TYPE ST_ServoMove :
STRUCT
	Name : STRING(Param_Servo.DESCRIPTION_LEN) := 'Actuator'; //Name visualized on UI
	AdvanceFeedback_Used : BOOL;      //TRUE if advanced state feedback is used  
	RetractFeedback_Used  : BOOL;      //TRUE if retracted state feedback is used  
	AdvanceFeedbackTimeoutError : TIME; // How long we wait to see advanced feedback before we raise timeout error; 0 if not used
	RetractFeedbackTimeoutError : TIME; // How long we wait to see retracted feedback before we raise timeout error; 0 if not used
	SimFeedback_Advance_TimeElapsed : TIME; //If we do not use Advanced Feedback, serves as simulation delay after Advance Output is Set
	SimFeedback_Retract_TimeElapsed : TIME; //If we do not use Retracted Feedback, serves as simulation delay after Advance Output is Set
END_STRUCT
END_TYPE

(* stored: Version 1.1.0.1, ProductVersion 3.1.4024.12
   DUT ST_ServoMove: Id {9a4051d5-0a8d-46c1-bb2d-34723daa6dfb} *)
